INTERFACE I_ParameterAddedEvent EXTENDS I_Event

PROPERTY PUBLIC TargetParameter : I_Parameter
GET
END_GET
END_PROPERTY

END_INTERFACE

(* stored: Version 1.1.0.1, ProductVersion 3.1.4024.12
   Itf I_ParameterAddedEvent: Id {8c23deb0-2d4b-49a2-b5cf-d2f917c264f6}
   Property TargetParameter: Id {82403ab7-23ac-437d-9d73-e41f90411bcb}
   Get Get: Id {6b33cfed-1029-4a7a-9d83-b6454db88557} *)
